PROGRAM ParameterEstimation
VAR
	//Inputs
	i1_raw, i2_raw, i3_raw	AT%I*: 					UINT;
	vX, vY, vTheta			AT%I*:					LREAL;
	robotPose				AT%I*:					RobotPose;
	
	state:											INT := 1;
	cnt:											INT := 0;
	
	Tsample:										REAL := 0.01;
	vmess:											LREAL:= 400;
	tmess:											REAL:=3;
	cnt_max:										INT;
	vTmp:											LREAL;
	
	//camera
	startX, startY, startTheta:						REAL;
	endX, endY, endTheta:							REAL;
	
	//odometrie
	odoX, odoY, odoTheta:							REAL := 0;
	
	//Outputs
	vout					AT%Q*:					LREAL;
	i1,i2,i3 				AT%Q*:					INT;	
	xErr, yErr, thetaErr    AT%Q*:					REAL;	
END_VAR

// Ströme umrechnen

i1 := UINT_TO_INT(i1_raw);
i2 := UINT_TO_INT(i2_raw);
i3 := UINT_TO_INT(i3_raw);


//Statemaschien Kovarianzvermessung
cnt_max := REAL_TO_INT(tmess/Tsample);

IF state = 1 THEN
	vout := vmess;
	
	IF cnt = 0 THEN
		odoX	:= 0;
		odoY	:= 0;
		odoTheta := 0;
		
		startX := robotPose.x;
		startY := robotPose.Y;
		startTheta := robotPose.Theta;
		
		xErr := (robotPose.x - startX) - odoX;
		yErr := (robotPose.y - startY) - odoY;
		thetaErr := (robotPose.Theta - startTheta) - odoTheta;
	ELSE
		cnt := cnt +1;
	END_IF
	
	IF cnt > cnt_max/3 THEN
		state := 2;cnt 	:= 0;
	END_IF
END_IF

IF state = 2 THEN
	
	odoX := odoX + vX*Tsample;	
	odoY := odoY + vY*Tsample;
	odoTheta := odoTheta + vTheta*Tsample;
	
	cnt := cnt + 1;
	IF cnt > cnt_max THEN
		state := 3; vout:= 0; cnt := 0;
	END_IF
END_IF

IF state = 3 THEN
	vout := -vmess;
	IF cnt = 0 THEN
		xErr := (robotPose.x - startX) - odoX;
		yErr := (robotPose.y - startY) - odoY;
		thetaErr := (robotPose.Theta - startTheta) - odoTheta;
		
		startX := robotPose.x;
		startY := robotPose.Y;
		startTheta := robotPose.Theta;
		
		odoX	:= 0;
		odoY	:= 0;
		odoTheta := 0;
		cnt := 1;
	ELSE
		cnt := cnt +1;
	END_IF
	
	IF cnt > cnt_max/3 THEN
		state := 4;cnt	:= 0;
	END_IF
END_IF

IF state = 4 THEN
	
	odoX := odoX + vX*Tsample;	
	odoY := odoY + vY*Tsample;
	odoTheta := odoTheta + vTheta*Tsample;

	cnt := cnt + 1;
	IF cnt > cnt_max THEN
		state := 1;vout := 0; cnt := 0;
	END_IF
END_IF

END_PROGRAM

(* stored: Version 1.1.0.1, ProductVersion 3.1.4024.11
   POU ParameterEstimation: Id {4296fb5a-753c-4dff-8f25-ad355e984a66}, SpecialFunc None *)
